(* PLC project Blank Project, Blank Blank 1.0 *)
(* stored: creationDateTime 2016-05-18T21:14:07, modificationDateTime 2023-05-02T10:20:21 *)

PROGRAM OverCurrent_FDR
  VAR
    Short_Circuit_FDR1 : BOOL;
    Short_Circuit_FDR2 : BOOL;
    Short_Circuit_FDR3 : BOOL;
    Short_Circuit_FDR4 : BOOL;
    Short_Circuit_22BUS1 : BOOL;
    Short_Circuit_22BUS2 : BOOL;
  END_VAR
  VAR
    Open_CB1_22KV AT %QX0.0 : BOOL;
    Open_CB2_22KV AT %QX0.1 : BOOL := TRUE;
    Open_CB3_22KV AT %QX0.2 : BOOL;
    Open_CB_FDR1 AT %QX0.3 : BOOL;
    Open_CB_FDR2 AT %QX0.4 : BOOL;
    Open_CB_FDR3 AT %QX0.5 : BOOL;
    Open_CB_FDR4 AT %QX0.6 : BOOL;
    Reset_All_CB AT %IX0.0 : BOOL;
    Current_22BUS1 AT %IW0 : INT;
    Current_22BUS2 AT %IW1 : INT;
    Current_22BUS3 AT %IW2 : INT;
    Current_FDR1 AT %IW3 : INT;
    Current_FDR2 AT %IW4 : INT;
    Current_FDR3 AT %IW5 : INT;
    Current_FDR4 AT %IW6 : INT;
    Fault_on_22BUS1_Current AT %IW7 : INT;
    Fault_on_22BUS2_Current AT %IW8 : INT;
    Fault_on_FDR1_Current AT %IW9 : INT;
    Fault_on_FDR2_Current AT %IW10 : INT;
    Fault_on_FDR3_Current AT %IW11 : INT;
    Fault_on_FDR4_Current AT %IW12 : INT;
  END_VAR
  VAR CONSTANT
    Threshold : INT := 500;
  END_VAR

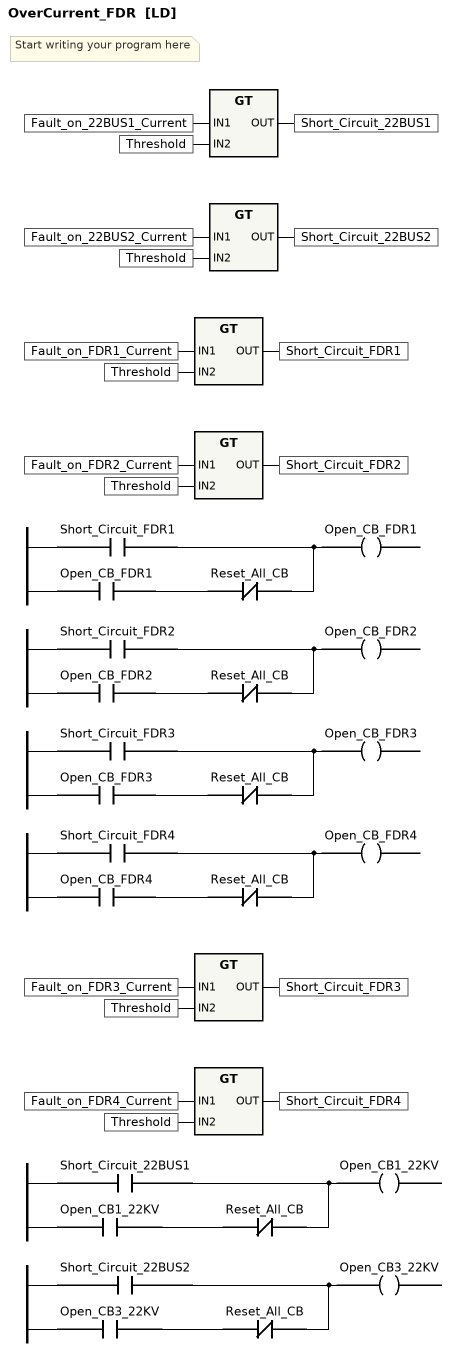
(* LD diagram, written out as Structured Text *)
(* Start writing your program here *)
Open_CB1_22KV := Open_CB1_22KV AND NOT Reset_All_CB OR Short_Circuit_22BUS1;
Short_Circuit_22BUS1 := Fault_on_22BUS1_Current > Threshold;
Open_CB3_22KV := Short_Circuit_22BUS2 OR Open_CB3_22KV AND NOT Reset_All_CB;
Short_Circuit_22BUS2 := Fault_on_22BUS2_Current > Threshold;
Open_CB_FDR1 := Short_Circuit_FDR1 OR Open_CB_FDR1 AND NOT Reset_All_CB;
Short_Circuit_FDR1 := Fault_on_FDR1_Current > Threshold;
Open_CB_FDR2 := Open_CB_FDR2 AND NOT Reset_All_CB OR Short_Circuit_FDR2;
Short_Circuit_FDR2 := Fault_on_FDR2_Current > Threshold;
Open_CB_FDR3 := Open_CB_FDR3 AND NOT Reset_All_CB OR Short_Circuit_FDR3;
Short_Circuit_FDR3 := Fault_on_FDR3_Current > Threshold;
Open_CB_FDR4 := Short_Circuit_FDR4 OR Open_CB_FDR4 AND NOT Reset_All_CB;
Short_Circuit_FDR4 := Fault_on_FDR4_Current > Threshold;
END_PROGRAM

CONFIGURATION Config0
  RESOURCE Res0 ON PLC
    TASK TaskMain(INTERVAL := T#10ms, PRIORITY := 0);
    PROGRAM Inst0 WITH TaskMain : OverCurrent_FDR;
  END_RESOURCE
END_CONFIGURATION
